(* IEC 61131-3 sources: volt/packages/volt-lsp-iec/test-corpus/lenze-mid/Device/Plc Logic/Application/Library Manager/CmpBinTagUtilIec, 37 files *)

(* ---- BTAGALIGNMENT.dut ---- *)
TYPE BTAGALIGNMENT :
STRUCT
	UIMODULUS : UINT;
	UIREMAINDER : UINT;
END_STRUCT
END_TYPE

(* ---- BTAGELEMENTTYPE.dut ---- *)
TYPE BTAGELEMENTTYPE :
(
	STARTTAG := 0,
	ENDTAG := 1,
	EOF := 2
);
END_TYPE

(* ---- TESTCASES.dut ---- *)
TYPE TESTCASES :
(
	CREATEWRITER,
	WRITERINIT,
	STARTTAG1,
	STARTTAG2,
	STARTTAG3,
	STARTTAG4,
	APPENDBLOB1,
	APPENDBLOB2,
	APPENDBLOB3,
	APPENDBLOB4,
	APPENDFILLBYTES1,
	APPENDFILLBYTES2,
	ENDTAG1,
	ENDTAG2,
	ENDTAG3,
	ENDTAG4,
	FINISH1,
	FINISH2,
	FINISH3,
	DESTROYWRITER,
	CREATEREADER,
	READERINIT,
	DESTROYREADER,
	PEEK1,
	PEEK2,
	DATATAG1,
	DATATAG2,
	GETTAGID1,
	GETTAGID2,
	GETTAGID3,
	GETTAGLEN1,
	GETTAGLEN2,
	MOVENEXT1,
	MOVENEXT2,
	MOVENEXT3,
	MOVENEXT4,
	MOVENEXT5,
	MOVENEXT6,
	GETCONTENT1,
	GETCONTENT2,
	MAXNUM
);
END_TYPE

(* ---- BTAGALIGNMENTS.gvl ---- *)
VAR_GLOBAL
	ALIGN42 : BTagAlignment := STRUCT(uiModulus := 4, uiRemainder := 2);
	ALIGN40 : BTagAlignment := STRUCT(uiModulus := 4, uiRemainder := 0);
END_VAR

(* ---- RETURNVALUES.gvl ---- *)
VAR_GLOBAL
	ERR_OK : UDINT := 16#0;
	ERR_FAILED : UDINT := 16#1;
	ERR_PARAMETER : UDINT := 16#2;
	ERR_NOTIMPLEMENTED : UDINT := 16#C;
	ERR_NOMEMORY : UDINT := 16#11;
	ERR_BTAG_TAGOVERLAP : UDINT := 16#400;
	ERR_BTAG_BUFFEROVERRUN : UDINT := 16#401;
	ERR_BTAG_MAXNESTINGDEPTH : UDINT := 16#402;
	ERR_BTAG_NOTAG : UDINT := 16#403;
	ERR_BTAG_NODATATAG : UDINT := 16#404;
	ERR_BTAG_NOCONTAINERTAG : UDINT := 16#405;
	ERR_BTAG_NOTTOPLEVEL : UDINT := 16#406;
	ERR_BTAG_ALIGNMENT : UDINT := 16#407;
	INVALID_HANDLE : __UXINT := RTS_INVALID_HANDLE;
END_VAR

(* ---- BTAGREADERCREATE.pou ---- *)
FUNCTION BTAGREADERCREATE : RTS_IEC_HANDLE
VAR_INPUT
	PBUFFER : POINTER TO BYTE;
	DWSIZE : DWORD;
	PRESULT : POINTER TO RTS_IEC_RESULT;
END_VAR
END_FUNCTION

(* ---- BTAGREADERCREATEDYNAMIC.pou ---- *)
FUNCTION BTAGREADERCREATEDYNAMIC : RTS_IEC_HANDLE
VAR_INPUT
	PRESULT : POINTER TO RTS_IEC_RESULT;
END_VAR
END_FUNCTION

(* ---- BTAGREADERDESTROY.pou ---- *)
FUNCTION BTAGREADERDESTROY : RTS_IEC_RESULT
VAR_INPUT
	HREADER : RTS_IEC_HANDLE;
END_VAR
END_FUNCTION

(* ---- BTAGREADERGETCOMPLEXCONTENT.pou ---- *)
FUNCTION BTAGREADERGETCOMPLEXCONTENT : RTS_IEC_RESULT
VAR_INPUT
	HREADER : RTS_IEC_HANDLE;
	PPBUFFER : POINTER TO POINTER TO BYTE;
	PULSIZE : POINTER TO UDINT;
END_VAR
END_FUNCTION

(* ---- BTAGREADERGETCONTENT.pou ---- *)
FUNCTION BTAGREADERGETCONTENT : RTS_IEC_RESULT
VAR_INPUT
	HREADER : RTS_IEC_HANDLE;
	PPBUFFER : POINTER TO POINTER TO BYTE;
	PULSIZE : POINTER TO UDINT;
END_VAR
END_FUNCTION

(* ---- BTAGREADERGETSTRING.pou ---- *)
FUNCTION BTAGREADERGETSTRING : RTS_IEC_RESULT
VAR_INPUT
	HREADER : RTS_IEC_HANDLE;
	PPBUFFER : POINTER TO POINTER TO BYTE;
	PULSIZE : POINTER TO UDINT;
	BADDENDOFSTRING : BOOL;
END_VAR
END_FUNCTION

(* ---- BTAGREADERGETTAGID.pou ---- *)
FUNCTION BTAGREADERGETTAGID : RTS_IEC_RESULT
VAR_INPUT
	HREADER : RTS_IEC_HANDLE;
	PULTAGID : POINTER TO UDINT;
END_VAR
END_FUNCTION

(* ---- BTAGREADERGETTAGLEN.pou ---- *)
FUNCTION BTAGREADERGETTAGLEN : RTS_IEC_RESULT
VAR_INPUT
	HREADER : RTS_IEC_HANDLE;
	PULTAGLEN : POINTER TO UDINT;
END_VAR
END_FUNCTION

(* ---- BTAGREADERINIT.pou ---- *)
FUNCTION BTAGREADERINIT : RTS_IEC_RESULT
VAR_INPUT
	HREADER : RTS_IEC_HANDLE;
	PBUFFER : POINTER TO BYTE;
	DWBUFFERSIZE : DWORD;
END_VAR
END_FUNCTION

(* ---- BTAGREADERISDATATAG.pou ---- *)
FUNCTION BTAGREADERISDATATAG : RTS_IEC_RESULT
VAR_INPUT
	HREADER : RTS_IEC_HANDLE;
	PBDATATAG : POINTER TO BOOL;
END_VAR
END_FUNCTION

(* ---- BTAGREADERMOVENEXT.pou ---- *)
FUNCTION BTAGREADERMOVENEXT : RTS_IEC_RESULT
VAR_INPUT
	HREADER : RTS_IEC_HANDLE;
	PNELEMENTTYPE : POINTER TO BTagElementType;
END_VAR
END_FUNCTION

(* ---- BTAGREADERPEEKNEXT.pou ---- *)
FUNCTION BTAGREADERPEEKNEXT : BTagElementType
VAR_INPUT
	HREADER : RTS_IEC_HANDLE;
END_VAR
END_FUNCTION

(* ---- BTAGREADERSKIPCONTENT.pou ---- *)
FUNCTION BTAGREADERSKIPCONTENT : RTS_IEC_RESULT
VAR_INPUT
	HREADER : RTS_IEC_HANDLE;
END_VAR
END_FUNCTION

(* ---- BTAGSWAPHEADER.pou ---- *)
FUNCTION BTAGSWAPHEADER : DWORD
VAR_INPUT
	PHEADERTAG : POINTER TO DWORD;
	BSWAP : DINT;
END_VAR
END_FUNCTION

(* ---- BTAGWRITERAPPENDBLOB.pou ---- *)
FUNCTION BTAGWRITERAPPENDBLOB : RTS_IEC_RESULT
VAR_INPUT
	HWRITER : RTS_IEC_HANDLE;
	PDATA : POINTER TO BYTE;
	DWDATASIZE : DWORD;
END_VAR
END_FUNCTION

(* ---- BTAGWRITERAPPENDDUMMYBYTES.pou ---- *)
FUNCTION BTAGWRITERAPPENDDUMMYBYTES : RTS_IEC_RESULT
VAR_INPUT
	HWRITER : RTS_IEC_HANDLE;
	BTFILL : BYTE;
	ULCOUNT : DWORD;
END_VAR
END_FUNCTION

(* ---- BTAGWRITERAPPENDFILLBYTES.pou ---- *)
FUNCTION BTAGWRITERAPPENDFILLBYTES : RTS_IEC_RESULT
VAR_INPUT
	HWRITER : RTS_IEC_HANDLE;
	BTFILL : BYTE;
	ALIGNMENT : BTagAlignment;
END_VAR
END_FUNCTION

(* ---- BTAGWRITERAPPENDRAW.pou ---- *)
FUNCTION BTAGWRITERAPPENDRAW : RTS_IEC_RESULT
VAR_INPUT
	HWRITER : RTS_IEC_HANDLE;
	PPDATA : POINTER TO POINTER TO BYTE;
	DWSIZE : DWORD;
END_VAR
END_FUNCTION

(* ---- BTAGWRITERAPPENDWSTRING.pou ---- *)
FUNCTION BTAGWRITERAPPENDWSTRING : RTS_IEC_RESULT
VAR_INPUT
	HWRITER : RTS_IEC_HANDLE;
	WSZSTRING : REFERENCE TO WSTRING;
END_VAR
END_FUNCTION

(* ---- BTAGWRITERCREATE.pou ---- *)
FUNCTION BTAGWRITERCREATE : RTS_IEC_HANDLE
VAR_INPUT
	PBUFFER : POINTER TO BYTE;
	DWSIZE : DWORD;
	PRESULT : POINTER TO RTS_IEC_RESULT;
END_VAR
END_FUNCTION

(* ---- BTAGWRITERCREATEDYNAMIC.pou ---- *)
FUNCTION BTAGWRITERCREATEDYNAMIC : RTS_IEC_HANDLE
VAR_INPUT
	PRESULT : POINTER TO RTS_IEC_RESULT;
END_VAR
END_FUNCTION

(* ---- BTAGWRITERCREATESAVEPOINT.pou ---- *)
FUNCTION BTAGWRITERCREATESAVEPOINT : RTS_IEC_HANDLE
VAR_INPUT
	HWRITER : RTS_IEC_HANDLE;
	PDATA : POINTER TO BYTE;
	DWDATASIZE : DWORD;
	PRESULT : POINTER TO RTS_IEC_RESULT;
END_VAR
END_FUNCTION

(* ---- BTAGWRITERCREATESAVEPOINTDYNAMIC.pou ---- *)
FUNCTION BTAGWRITERCREATESAVEPOINTDYNAMIC : RTS_IEC_HANDLE
VAR_INPUT
	HWRITER : RTS_IEC_HANDLE;
	PRESULT : POINTER TO RTS_IEC_RESULT;
END_VAR
END_FUNCTION

(* ---- BTAGWRITERDESTROY.pou ---- *)
FUNCTION BTAGWRITERDESTROY : RTS_IEC_RESULT
VAR_INPUT
	HWRITER : RTS_IEC_HANDLE;
END_VAR
END_FUNCTION

(* ---- BTAGWRITERDESTROYSAVEPOINT.pou ---- *)
FUNCTION BTAGWRITERDESTROYSAVEPOINT : RTS_IEC_RESULT
VAR_INPUT
	HSAVEPOINT : RTS_IEC_HANDLE;
END_VAR
END_FUNCTION

(* ---- BTAGWRITERENDTAG.pou ---- *)
FUNCTION BTAGWRITERENDTAG : RTS_IEC_RESULT
VAR_INPUT
	HWRITER : RTS_IEC_HANDLE;
	UDITAGID : UDINT;
END_VAR
END_FUNCTION

(* ---- BTAGWRITERFINISH.pou ---- *)
FUNCTION BTAGWRITERFINISH : RTS_IEC_RESULT
VAR_INPUT
	HWRITER : RTS_IEC_HANDLE;
	PPBUFFER : POINTER TO POINTER TO BYTE;
	PUISIZE : POINTER TO UDINT;
END_VAR
END_FUNCTION

(* ---- BTAGWRITERINIT.pou ---- *)
FUNCTION BTAGWRITERINIT : RTS_IEC_RESULT
VAR_INPUT
	HWRITER : RTS_IEC_HANDLE;
	PBUFFER : POINTER TO BYTE;
	DWBUFFERSIZE : DWORD;
END_VAR
END_FUNCTION

(* ---- BTAGWRITERINIT2.pou ---- *)
FUNCTION BTAGWRITERINIT2 : RTS_IEC_RESULT
VAR_INPUT
	HWRITER : RTS_IEC_HANDLE;
	PBUFFER : POINTER TO BYTE;
	DWBUFFERSIZE : DWORD;
	BSWAP : DINT;
END_VAR
END_FUNCTION

(* ---- BTAGWRITERRESTORESAVEPOINT.pou ---- *)
FUNCTION BTAGWRITERRESTORESAVEPOINT : RTS_IEC_RESULT
VAR_INPUT
	HWRITER : RTS_IEC_HANDLE;
	HSAVEPOINT : RTS_IEC_HANDLE;
END_VAR
END_FUNCTION

(* ---- BTAGWRITERSTARTTAG.pou ---- *)
FUNCTION BTAGWRITERSTARTTAG : RTS_IEC_RESULT
VAR_INPUT
	HWRITER : RTS_IEC_HANDLE;
	UDITAGID : UDINT;
	ALIGNMENT : BTagAlignment;
	UDIMINLENGTHSIZE : UDINT;
END_VAR
END_FUNCTION

(* ---- BTAGWRITERSWITCHBUFFER.pou ---- *)
FUNCTION BTAGWRITERSWITCHBUFFER : RTS_IEC_RESULT
VAR_INPUT
	HWRITER : RTS_IEC_HANDLE;
	PNEWBUFFER : POINTER TO BYTE;
	DWNEWBUFFERSIZE : DWORD;
	PPOLDBUFFER : POINTER TO POINTER TO BYTE;
END_VAR
END_FUNCTION
